TYPE EL5102_ENC_ControlChannel :
STRUCT
	{attribute addProperty Name "Control"}
	Control AT %Q* : EL5102_Control;
	{attribute addProperty Name "Set counter value"}
	SetCounterValue AT %Q* : UDINT;
END_STRUCT
END_TYPE

(* stored: Version 1.1.0.1, ProductVersion 3.1.4024.9
   DUT EL5102_ENC_ControlChannel: Id {dab063e5-f22b-05ca-3f8e-b89566a5ec29} *)
